FUNCTION_BLOCK INTERNAL FB_HasCoinState IMPLEMENTS I_State
VAR_INPUT
END_VAR
VAR_OUTPUT
END_VAR
VAR
	pMachine : POINTER TO FB_Machine;
END_VAR

METHOD CustomerTakesCoin : BOOL
END_METHOD

METHOD CustomerTakesProduct : BOOL
END_METHOD

PROPERTY Description : STRING
GET
Description := 'Has Coin';
END_GET
END_PROPERTY

METHOD FB_init : BOOL
VAR_INPUT
	bInitRetains : BOOL; // if TRUE, the retain variables are initialized (warm start / cold start)
	bInCopyCode : BOOL;  // if TRUE, the instance afterwards gets moved into the copy code (online change)
	pMachine : POINTER TO FB_Machine;
END_VAR
THIS^.pMachine := pMachine;
END_METHOD

METHOD InsertCoin : BOOL
END_METHOD

METHOD PressButton : BOOL
IF (THIS^.pMachine^.nProducts > 0) THEN
	THIS^.pMachine^.SetProducts(THIS^.pMachine^.nProducts - 1);
	ADSLOGSTR(ADSLOG_MSGTYPE_HINT, 'Customer has pressed the button. Output product.', '');
	pMachine^.SetState(pMachine^.ProductEjectedState);
ELSE				
	ADSLOGSTR(ADSLOG_MSGTYPE_HINT, 'Customer has pressed the button. No more products. Return coin.', '');
	pMachine^.SetState(pMachine^.CoinEjectedState);
END_IF
END_METHOD

END_FUNCTION_BLOCK

(* stored: Version 1.1.0.1, ProductVersion 3.1.4022.12
   POU FB_HasCoinState: Id {4542327b-fad5-4127-93a5-9d754c5837fa}, SpecialFunc None
   Method CustomerTakesCoin: Id {07079302-8fd3-40ec-9e46-e23b26f356a3}
   Method CustomerTakesProduct: Id {e30930e8-d194-4d35-a0ed-41c3b52ab562}
   Property Description: Id {92a2c821-977c-4c79-a9fa-fa2bcd58c838}
   Get Get: Id {bd2e2ec5-7306-4b52-acb5-68a1282ac942}
   Method FB_init: Id {46bc79d9-3ab7-4dcb-8db7-f56fc6b87ff7}
   Method InsertCoin: Id {6cce552f-84aa-4529-92c1-362ac4c4dae2}
   Method PressButton: Id {e9153bdc-1d24-471d-a8bb-7326ab81bb1e} *)
